{attribute 'linkalways'} 
{attribute 'no_explicit_call' := 'This FB is a CLASS and must be accessed using methods or properties'}
{attribute 'enable_dynamic_creation'}
FUNCTION_BLOCK Node_F_VN_Threshold EXTENDS VisionNode
VAR
	ipSrcImage : _ITcVnImage;
    ipDestImage : _ITcVnImage;
    fThreshold : _LREAL(0.0);
    fMaxValue : _LREAL(0.0);
	eThresholdType : _ETcVnThresholdType(ETcVnThresholdType.TCVN_TT_BINARY);
    hrPrev : _HRESULT(S_OK);
	hresult : _HRESULT(S_OK);
END_VAR

METHOD PUBLIC  Clone : I_Node
VAR
	pNode : POINTER TO Node_F_VN_Threshold;
END_VAR
pNode := __NEW(Node_F_VN_Threshold);
Clone := pNode^;
END_METHOD

METHOD FB_init : BOOL
VAR_INPUT
	bInitRetains : BOOL; // if TRUE, the retain variables are initialized (warm start / cold start)
	bInCopyCode : BOOL;  // if TRUE, the instance afterwards gets moved into the copy code (online change)
END_VAR
AddInput('ipSrcImage', ipSrcImage);
AddParameter('fThreshold', fThreshold);
AddParameter('fMaxValue', fMaxValue);
AddParameter('eThresholdType', eThresholdType);
AddInput('hrPrev', hrPrev);
AddOutput('ipDestImage', ipDestImage);
AddOutput('hresult',hresult);
END_METHOD

METHOD PROTECTED OnExecute
hresult.Value := F_VN_Threshold(
	ipSrcImage := ipSrcImage.Value, 
	ipDestImage := ipDestImage.Value, 
	fThreshold := fThreshold.Value, 
	fMaxValue := fMaxValue.Value, 
	eThresholdType := eThresholdType.Value, 
	hrPrev := hrPrev.Value);
END_METHOD

METHOD PUBLIC PreExecutionCheck
VAR_INPUT
	Check : I_PreExecutionChecks;
END_VAR
VAR
    dynamicThresholding : BOOL;
    pixelFormat : TcVnPixelFormat;
END_VAR
Check.IsTrue(ipSrcImage.IsValid, 'ipSrcImage must contain an image');

CASE eThresholdType.Value OF
    TCVN_TT_OTSU_BINARY,
    TCVN_TT_OTSU_BINARY_INV,
    TCVN_TT_OTSU_TRUNC,
    TCVN_TT_OTSU_TOZERO,
    TCVN_TT_OTSU_TOZERO_INV,
    TCVN_TT_TRIANGLE_BINARY,
    TCVN_TT_TRIANGLE_BINARY_INV,
    TCVN_TT_TRIANGLE_TRUNC,
    TCVN_TT_TRIANGLE_TOZERO,
    TCVN_TT_TRIANGLE_TOZERO_INV :
        dynamicThresholding := TRUE;
END_CASE

IF dynamicThresholding THEN
    Check.IsTrue(ipSrcImage.HasChannelCount(1), 'ipSrcImage must have 1 channel when using dynamic thresholding');
    Check.IsTrue(ipSrcImage.IsPixelDepth(8), 'ipSrcImage must have 8 bit pixel depth when using dynamic thresholding');
ELSE
    Check.IsTrue((ipSrcImage.HasChannelCount(1) OR ipSrcImage.HasChannelCount(3)), 'ipSrcImage must have 1 or 3 channels');
END_IF

ipSrcImage.TryGetPixelFormat(pixelFormat);
Check.IsTrue(IsMaxValueCompatibleWithPixelDepth(fMaxValue.Value, pixelFormat.nElementSize), 'fMaxValue is not compatible with pixel depth');
END_METHOD

END_FUNCTION_BLOCK

(* stored: Version 1.1.0.1, ProductVersion 3.1.4024.15
   POU Node_F_VN_Threshold: Id {4c21a7fe-dcfa-022e-3e68-912bd9a18686}, SpecialFunc None
   Folder Constructor: Id {e7e744ce-064d-03c2-1e48-e04623a658cd}
   Method Clone: Id {0178e9bd-d193-0bf1-1afc-6efdcc11dd60}
   Method FB_init: Id {80e5081c-306e-0c22-1443-531957b65003}
   Method OnExecute: Id {34fdcd61-bc23-0040-09c7-acdd0eb6cb2c}
   Method PreExecutionCheck: Id {0ecf4454-3e18-059b-112e-62ddfae38d27} *)
